Staubli VAL3: computeFrame.pgx

public program computeFrame(num x_nNewFrame)
begin
end
